// TIA Portal V20 export
TYPE "UDT_RFID_STN_Data"
   STRUCT
      Station_Task : Byte;   // 工位建造状态（0:未完成 1:接受 2:拒绝）
      TASK_01 : Byte;   // 任务1状态（0:未完成 1:接受 2:拒绝）
      TASK_02 : Byte;   // 任务2状态（0:未完成 1:接受 2:拒绝）
      TASK_03 : Byte;   // 任务3状态（0:未完成 1:接受 2:拒绝）
      TASK_04 : Byte;   // 任务4状态（0:未完成 1:接受 2:拒绝）
      TASK_05 : Byte;   // 任务5状态（0:未完成 1:接受 2:拒绝）
      TASK_06 : Byte;   // 任务6状态（0:未完成 1:接受 2:拒绝）
      TASK_07 : Byte;   // 任务7状态（0:未完成 1:接受 2:拒绝）
      TASK_08 : Byte;   // 任务8状态（0:未完成 1:接受 2:拒绝）
      TASK_09 : Byte;   // 任务9状态（0:未完成 1:接受 2:拒绝）
   END_STRUCT;
END_TYPE
